(* CoDeSys 2.3.9.44 project: IEC61131.PRO *)
(* Libraries: standard.lib 10.8.21 12:06:01, C3_ObjectDirT30.lib 10.8.21 12:06:01, C3_FunctionsT30.lib 10.8.21 12:06:01, C3_Debug.lib 10.8.21 12:06:00, C3_PLCOpenT30.lib 10.8.21 12:06:01 *)

(* POU PLC_PRG, ST *)
PROGRAM PLC_PRG

VAR CONSTANT
	CPXenable1: INT := 1;
	CPXenable2: INT := 2;
	CPXstop: INT := 9;
	CPXreset: INT := 10;
	CPXhome: INT := 11;
	CPXposabs: INT := 12;
	CPXposrel: INT := 13;
	CPXdisable: INT := 14;
	CPXoutput: INT := 15;

	CPXIO0: INT := 0;
	CPXIO1: INT := 1;
	CPXIO2: INT := 2;
	CPXIO3: INT := 3;

	CMD_None: INT := 0;
	CMD_Reset: INT := 1;
	CMD_Stop: INT := 2;
	CMD_Home: INT := 3;
	CMD_MoveAbsolute: INT := 4;
	CMD_MoveRelative: INT := 5;
	CMD_Done: INT := 100;
END_VAR

VAR
	MCPower: MC_Power;
	MCStop: MC_Stop;
	MCReset: MC_Reset;
	MCHome: MC_Home;
	MCMoveAbsolute: MC_MoveAbsolute;
	MCMoveRelative: MC_MoveRelative;
	Inputs: C3_Input;
	Outputs: C3_Output;
	AosOutputs: C3_IOAddition_0;
	cmd: INT;
	cmdlast: INT := 0;
	runcmd: INT := 0;
	startcmd: INT;
	halfwindow: REAL;
	diff: REAL;
	enable: BOOL := 0;

	IO_point_address: INT := 0;
	IO_point_value: INT := 0;
	IO_point_state: BOOL := FALSE;

	SIM_INPUT_4: BOOL := FALSE;
END_VAR
(* Read signals AND command registers *)
inputs();
startcmd := 0;
cmd := C3Array.Col05_Row01;
IO_point_address := C3Array.Col05_Row06;
IO_point_value := C3Array.Col05_Row07;

(* Update device state *)
C3Plus.DeviceState_Statusword_2.0 := Outputs.O0;
C3Plus.DeviceState_Statusword_2.1 := Outputs.O1;
C3Plus.DeviceState_Statusword_2.2 := Outputs.O2;
C3Plus.DeviceState_Statusword_2.3 := Outputs.O3;

C3Plus.DeviceState_Statusword_2.4 := Inputs.I0;
C3Plus.DeviceState_Statusword_2.5 := Inputs.I1;
C3Plus.DeviceState_Statusword_2.6 := Inputs.I2;
C3Plus.DeviceState_Statusword_2.7 := Inputs.I3;
C3Plus.DeviceState_Statusword_2.8 := Inputs.I4;
C3Plus.DeviceState_Statusword_2.9 := Inputs.I5;
C3Plus.DeviceState_Statusword_2.10 := Inputs.I6;
C3Plus.DeviceState_Statusword_2.11 := Inputs.I7;

C3Plus.DeviceState_Statusword_2.12 := MCPower.Enable;
C3Plus.DeviceState_Statusword_2.13 := C3Plus.ErrorHistory_LastError;

IF C3Array.Col05_Row05 = 1 THEN
	SIM_INPUT_4 := TRUE;
ELSE
	SIM_INPUT_4 := FALSE;
END_IF

(* Check Enable-signal *)
IF cmdlast = CPXenable1 AND cmd = CPXenable2 THEN
	enable := TRUE;
END_IF
cmdlast := cmd;
IF Inputs.I2 = TRUE AND inputs.I3 = TRUE THEN
	IF enable = TRUE THEN
		MCPower.Enable := TRUE;
		C3Array.Col05_Row01 := 0;			(* No command *)
		enable := FALSE;
	END_IF
ELSE
	MCPower.Enable := FALSE;
END_IF

(* Check Reset command *)
IF cmd = CPXreset THEN
	CASE runcmd OF
		CMD_Done, CMD_Reset:;
	ELSE
		startcmd := CMD_Reset;
		MCReset.Execute := TRUE;
	END_CASE
END_IF

(* Check Disable command *)
IF cmd = CPXdisable THEN
		MCStop.Execute := FALSE;
		MCHome.Execute := FALSE;
		MCMoveAbsolute.Execute := FALSE;
		MCMoveRelative.Execute := FALSE;
		MCPower.Enable := FALSE;
		startcmd := CMD_Done;
END_IF

(* Check Output commands *)
IF cmd = CPXoutput THEN
	IF IO_point_value = 0 OR IO_point_value = 1 THEN
		CASE IO_point_address OF
			0:
				Outputs.O0 := INT_TO_BOOL(IO_point_value);
			1:
				Outputs.O1 := INT_TO_BOOL(IO_point_value);
			2:
				Outputs.O2 := INT_TO_BOOL(IO_point_value);
			3:
				Outputs.O3 := INT_TO_BOOL(IO_point_value);
		END_CASE
	END_IF

	C3Array.Col05_Row06 := 0;
	C3Array.Col05_Row07 := 0;
	C3Array.Col05_Row01 := 0;
END_IF


(* Check Run-signal *)
IF inputs.I4 = TRUE OR SIM_INPUT_4 = TRUE THEN
	C3Array.Col04_Row01 := 1;				(* Confirm RUN *)
	IF runcmd = CMD_None OR cmd = CPXstop THEN
		CASE cmd OF
			CPXhome:
				startcmd := CMD_Home;
				MCHome.Position := C3Array.Col01_Row01;
				MCHome.Execute := TRUE;
			CPXposabs:
				startcmd := CMD_MoveAbsolute;
				MCMoveAbsolute.Position := C3Array.Col01_Row01;
				MCMoveAbsolute.Velocity := C3Array.Col02_Row01;
				MCMoveAbsolute.Acceleration := C3Array.Col06_Row01;
				MCMoveAbsolute.Deceleration := C3Array.Col07_Row01;
				MCMoveAbsolute.Jerk := C3Array.Col08_Row01;
				MCMoveAbsolute.JerkDecel := C3Array.Col09_Row01;
				MCMoveAbsolute.Execute := TRUE;
			CPXposrel:
				startcmd := CMD_MoveRelative;
				MCMoveRelative.Distance := C3Array.Col01_Row01;
				MCMoveRelative.Velocity := C3Array.Col02_Row01;
				MCMoveRelative.Acceleration := C3Array.Col06_Row01;
				MCMoveRelative.Deceleration := C3Array.Col07_Row01;
				MCMoveRelative.Jerk := C3Array.Col08_Row01;
				MCMoveRelative.JerkDecel := C3Array.Col09_Row01;
				MCMoveRelative.Execute := TRUE;
			CPXstop:
				startcmd := CMD_Stop;
				MCStop.Deceleration := C3Array.Col07_Row01;
				MCStop.Jerk := C3Array.Col09_Row01;
				MCStop.Execute := TRUE;
				MCHome.Execute := FALSE;
				MCMoveAbsolute.Execute := FALSE;
				MCMoveRelative.Execute := FALSE;
				C3Array.Col05_Row01 := 0;
			ELSE
				C3Array.Col05_Row01 := 0;	(* No command *)
		END_CASE
	END_IF
ELSE
	C3Array.Col04_Row01 := 0;				(* Confirm STOP *)
	IF MCPower.Status THEN
		CASE runcmd OF
			CMD_None, CMD_Done, CMD_Reset, CMD_Stop:;
		ELSE
			startcmd := CMD_Stop;
			MCStop.Deceleration := C3Array.Col07_Row01;
			MCStop.Jerk := C3Array.Col09_Row01;
			MCStop.Execute := TRUE;
			MCHome.Execute := FALSE;
			MCMoveAbsolute.Execute := FALSE;
			MCMoveRelative.Execute := FALSE;
		END_CASE
	END_IF
END_IF

(* Check Running commands *)
IF startcmd <> 0 THEN
	runcmd := startcmd;
ELSE
	CASE runcmd OF
		CMD_Reset:
			IF MCReset.Done OR MCReset.Error THEN
				MCReset.Execute := FALSE;
				runcmd := CMD_Done;
			END_IF
		CMD_Stop:
			IF NOT MCPower.Status OR MCStop.Done OR MCStop.Error THEN
				IF MCStop.Done THEN
					C3Array.Col01_Row02 := C3.StatusPosition_DemandValue;	(* Stop position *)
					C3Array.Col05_Row01 := 0;
				END_IF
				MCStop.Execute := FALSE;
				runcmd := CMD_Done;
			END_IF
		CMD_Home:
			IF MCHome.Done OR MCHome.CommandAborted OR MCHome.Error THEN
				IF MCHome.Done THEN
					C3Array.Col01_Row02 := C3.StatusPosition_DemandValue;	(* Stop position *)
				END_IF
				IF MCHome.CommandAborted THEN
					C3Array.Col03_Row01 := 1;								(* Command error *)
				END_IF
				MCHome.Execute := FALSE;
				runcmd := CMD_Done;
			END_IF
		CMD_MoveAbsolute:
			IF MCMoveAbsolute.Done OR MCMoveAbsolute.CommandAborted OR MCMoveAbsolute.Error THEN
				IF MCMoveAbsolute.Done THEN
					C3Array.Col01_Row02 := C3.StatusPosition_DemandValue;	(* Stop position *)
				END_IF
				IF MCMoveAbsolute.CommandAborted THEN
					C3Array.Col03_Row01 := 1;								(* Command error *)
				END_IF
				MCMoveAbsolute.Execute := FALSE;
				runcmd := CMD_Done;
			END_IF
		CMD_MoveRelative:
			IF MCMoveRelative.Done OR MCMoveRelative.CommandAborted OR MCMoveRelative.Error THEN
				IF MCMoveRelative.Done THEN
					C3Array.Col01_Row02 := C3.StatusPosition_DemandValue;	(* Stop position *)
				END_IF
				IF MCMoveRelative.CommandAborted THEN
					C3Array.Col03_Row01 := 1;								(* Command error *)
				END_IF
				MCMoveRelative.Execute := FALSE;
				runcmd := CMD_Done;
			END_IF
		CMD_Done:
			C3Array.Col05_Row01 := 0;		(* No command *)
			C3Array.Col05_Row05 := 0;
			runcmd := CMD_None;
	END_CASE
END_IF

IF C3Plus.ErrorHistory_LastError > 1 OR C3Array.Col03_Row01 > 0 THEN
	Outputs.O3 := TRUE;
ELSE
	Outputs.O3 := FALSE;
END_IF

(* Generate position pulses (ID-trig etc.) *)
(* Outputs.O0 := pulse(0, C3Array.Col01_Row10, C3Array.Col02_Row10, C3Array.Col03_Row10, C3Array.Col04_Row10);		(* ID-trig *) *)
AosOutputs.O0 := pulse(1, C3Array.Col01_Row11, C3Array.Col02_Row11, C3Array.Col03_Row11, C3Array.Col04_Row11);	(* Aos pulse 1 *)
AosOutputs.O1 := pulse(2, C3Array.Col01_Row12, C3Array.Col02_Row12, C3Array.Col03_Row12, C3Array.Col04_Row12);	(* Aos pulse 2 *)
AosOutputs.O2 := pulse(3, C3Array.Col01_Row13, C3Array.Col02_Row13, C3Array.Col03_Row13, C3Array.Col04_Row13);	(* Aos pulse 3 *)
AosOutputs.O3 := pulse(4, C3Array.Col01_Row14, C3Array.Col02_Row14, C3Array.Col03_Row14, C3Array.Col04_Row14);	(* Aos pulse 4 *)

Outputs();
AosOutputs(OutputEnable := TRUE);
MCPower(Axis := AXIS_REF_LocalAxis);
MCReset(Axis := AXIS_REF_LocalAxis);
MCStop(Axis := AXIS_REF_LocalAxis);
MCHome(Axis := AXIS_REF_LocalAxis);
MCMoveAbsolute(Axis := AXIS_REF_LocalAxis);
MCMoveRelative(Axis := AXIS_REF_LocalAxis);
END_PROGRAM

(* POU pulse, ST *)
FUNCTION pulse : BOOL
VAR_INPUT
	nr: INT;
	pos: REAL;
	pitch: REAL;
	window: INT;
	mode: INT;
END_VAR
VAR
	new: BOOL;
	diff: REAL;
	halfwindow: REAL;
END_VAR
(* Generate position pulse (ID-trig etc.) *)
IF window <> 0 THEN									(* Window ? *)
	diff := C3.StatusPosition_DemandValue - pos;	(* Current pos - Pulse pos *)
	halfwindow := window;							(* Window in 1/100 mm/deg *)
	halfwindow := halfwindow / 200.0;				(* Half window *)
	IF mode <> 0 THEN								(* Circular mode ? *)
		WHILE diff < -180.0 DO							(* Adjust diff to +/-180 *)
			diff := diff + 360.0;
		END_WHILE
		WHILE diff > 180.0 DO
			diff := diff - 360.0;
		END_WHILE
	END_IF
	new := FALSE;
	IF pitch < 0 THEN								(* Negative pitch *)
		IF diff + halfwindow < 0 THEN					(* Passed pulse ? *)
			pos := pos + pitch;								(* Add pitch *)
			new := TRUE;
		END_IF
	END_IF
	IF pitch > 0 THEN								(* Positive pitch *)
		IF diff - halfwindow > 0 THEN					(* Passed pulse ? *)
			pos := pos + pitch;								(* Add pitch *)
			new := TRUE;
		END_IF
	END_IF
	IF new = TRUE THEN
		CASE nr OF
			0: C3Array.Col01_Row10 := pos;
			1: C3Array.Col01_Row11 := pos;
			2: C3Array.Col01_Row12 := pos;
			3: C3Array.Col01_Row13 := pos;
			4: C3Array.Col01_Row14 := pos;
		END_CASE
	END_IF
	IF ABS(diff) <= halfwindow THEN					(* In pulse window ? *)
		pulse := TRUE;
		RETURN;
	END_IF
END_IF
pulse := FALSE;
END_FUNCTION
